{attribute 'qualified_only'}
VAR_GLOBAL
    (* 当前快速过程实际值。 *)
    stActual : ST_ProcessActual;
    (* 当前周期提取特征。 *)
    stFeatures : ST_ProcessFeatures;
    (* 四个工艺步骤的判据结果。 *)
    astStepCriterion : ARRAY[1..4] OF ST_StepCriterionResult;
    (* 最近完成的周期结果。 *)
    stLastCycleResult : ST_CycleResult;
END_VAR

(* stored: Version 1.1.0.1
   GVL GVL_Process: Id {C3100000-0000-4000-8000-000000000008} *)
